// TwinCAT 3 PLC project PLC
// ProgramVersion: 3.1.4024.0
// libraries:
//   EfficientIO ModbusTCP, * (EfficientIO)
//   Lynus Energy Basic, * (Lynus AG)
//   Lynus Persistent Data V1, * (Lynus AG)
//   Lynus Standards, * (Lynus AG)
//   Tc2_IoFunctions, * (Beckhoff Automation GmbH)
//   Tc2_Standard, * (Beckhoff Automation GmbH)
//   Tc2_System, * (Beckhoff Automation GmbH)
//   Tc3_IotBase, * (Beckhoff Automation GmbH)
//   Tc3_IPCDiag, * (Beckhoff Automation GmbH)
//   Tc3_Module, * (Beckhoff Automation GmbH)
// project tree:
//   / FastTask.TcTTO, MiddleTask.TcTTO, SlowTask.TcTTO
//   POUs/ prgComEffIO.TcPOU (excluded from build), prgComEffIO_1.TcPOU (excluded from build), prgEM.TcPOU, prgRWEffIO.TcPOU (not stored) (excluded from build), prgRWEffIO_1.TcPOU (excluded from build), prgTemperature.TcPOU, prgVarEffIO.TcPOU (not stored) (excluded from build), prgVarEffIO_1.TcPOU (excluded from build)
// real-time tasks:
//   TASK PlcTask: cycle T#10ms, priority 20, ADS port 350
//   TASK FastTask: cycle T#5ms, priority 19, ADS port 351
//   TASK MiddleTask: cycle T#10ms, priority 21, ADS port 352
//   TASK SlowTask: cycle T#20ms, priority 23, ADS port 353
// I/O:
//   DEVICE Gerät 2 (CX-BK)
//     Box 1 (CX-BK)
// variable links:
//   PLC/PLC Instance <-> Device 2 (CX-BK)/Box 1 (CX-BK)
//     PlcTask Inputs/prgEM.fbEM1.fbKL3403.byStateCH1 <-> Term 5 (KL3403)/Channel 1/Status
//     PlcTask Inputs/prgEM.fbEM1.fbKL3403.byStateCH2 <-> Term 5 (KL3403)/Channel 2/Status
//     PlcTask Inputs/prgEM.fbEM1.fbKL3403.byStateCH3 <-> Term 5 (KL3403)/Channel 3/Status
//     PlcTask Inputs/prgEM.fbEM1.fbKL3403.iDataInCH1 <-> Term 5 (KL3403)/Channel 1/Daten Ein
//     PlcTask Inputs/prgEM.fbEM1.fbKL3403.iDataInCH2 <-> Term 5 (KL3403)/Channel 2/Daten Ein
//     PlcTask Inputs/prgEM.fbEM1.fbKL3403.iDataInCH3 <-> Term 5 (KL3403)/Channel 3/Daten Ein
//     PlcTask Inputs/prgEM.fbKBusState.uiKBusState_OUT <-> Inputs/State
//     PlcTask Inputs/prgEM.stInData_22/iDataIn <-> Term 4 (KL3204)/Channel 1/Daten Ein
//     PlcTask Inputs/prgEM.stInData_23/iDataIn <-> Term 4 (KL3204)/Channel 2/Daten Ein
//     PlcTask Inputs/prgEM.stInData_22/iState <-> Term 4 (KL3204)/Channel 1/Status
//     PlcTask Inputs/prgEM.stInData_23/iState <-> Term 4 (KL3204)/Channel 2/Status
//     PlcTask Outputs/prgEM.fbEM1.fbKL3403.byCntrCH1 <-> Term 5 (KL3403)/Channel 1/Kontrolle
//     PlcTask Outputs/prgEM.fbEM1.fbKL3403.byCntrCH2 <-> Term 5 (KL3403)/Channel 2/Kontrolle
//     PlcTask Outputs/prgEM.fbEM1.fbKL3403.byCntrCH3 <-> Term 5 (KL3403)/Channel 3/Kontrolle
//     PlcTask Outputs/prgEM.stOutData_22/iCtrl <-> Term 4 (KL3204)/Channel 1/Kontrolle
//     PlcTask Outputs/prgEM.stOutData_23/iCtrl <-> Term 4 (KL3204)/Channel 2/Kontrolle
//     PlcTask Outputs/prgEM.stOutData_22/iDataOut <-> Term 4 (KL3204)/Channel 1/Daten Aus
//     PlcTask Outputs/prgEM.stOutData_23/iDataOut <-> Term 4 (KL3204)/Channel 2/Daten Aus

CONFIGURATION PLC
    RESOURCE PLC ON TwinCAT3
        TASK FastTask(INTERVAL := T#5ms, PRIORITY := 19);
        TASK MiddleTask(INTERVAL := T#10ms, PRIORITY := 21);
        TASK SlowTask(INTERVAL := T#20ms, PRIORITY := 23);
        PROGRAM prgEM WITH MiddleTask : prgEM;
        PROGRAM prgTemperature WITH MiddleTask : prgTemperature;
    END_RESOURCE
END_CONFIGURATION

// ---- POUs/prgEM.TcPOU
PROGRAM prgEM
VAR
	fbKBusState		: FB_K_Bus_State;
	fbEM1			: FB_EM_Beckhoff_KL3403;

END_VAR


fbKBusState(	uiKBusState_OUT=> , 
				b_Kbus_notOk=> , 
				word_ErrorCount=> );
//The mapping OF THIS FUNCTION must be linked with the KL3403 in the E/A Part
// KEBA CS
fbEM1(
	bEnable:= true, 
	bChannel1Invers:= FALSE,				//Invert power data when transformer are mounted upside down
	bChannel2Invers:= FALSE,			
	bChannel3Invers:= FALSE,
	uiCurrentTransformerRatioL1:= 100, //Transformer ratio on the secondary side
	uiCurrentTransformerRatioL2:= 100, 
	uiCurrentTransformerRatioL3:= 100, 
	uiKBusState_IN:= fbKBusState.uiKBusState_OUT, 
	stDataEMPower=> , 
	stDataEMCounter=> , 
	stDataEMPowerRealTime=> , 
	stDataEMCounterRealTime=> , 
	diNrOfEM_OUT=> );

END_PROGRAM

// ---- POUs/prgTemperature.TcPOU
PROGRAM prgTemperature
VAR
// Kanal 1
	fb_Config_1			: FB_KL320xConfig;
	stInData_1   		AT%I*		: ST_KL320xInData;
	stOutData_1		  	AT%Q*		: ST_KL320xOutData;
// Kanal 2
	fb_Config_2			: FB_KL320xConfig;
	stInData_2   		AT%I*		: ST_KL320xInData;
	stOutData_2  		AT%Q*		: ST_KL320xOutData;

END_VAR

	
	
fb_Config_1(
	bConfigurate:= , 
	bReadConfig:= , 
	iSetSensorType:= , 
	tTimeout:= , 
	bBusy=> , 
	bError=> , 
	iErrorId=> , 
	iState=> , 
	iDataIn=> , 
	iTerminalType=> , 
	iSpecialType=> , 
	iFirmwareVersion=> , 
	sDescription=> , 
	sSensorType=> , 
	bTwoWiredConnection=> , 
	stInData:= stInData_1, 
	stOutData:= stOutData_1);
	
fb_Config_2(
	bConfigurate:= , 
	bReadConfig:= , 
	iSetSensorType:= , 
	tTimeout:= , 
	bBusy=> , 
	bError=> , 
	iErrorId=> , 
	iState=> , 
	iDataIn=> , 
	iTerminalType=> , 
	iSpecialType=> , 
	iFirmwareVersion=> , 
	sDescription=> , 
	sSensorType=> , 
	bTwoWiredConnection=> , 
	stInData:= stInData_2, 
	stOutData:= stOutData_2);

END_PROGRAM

// ---- POUs/prgComEffIO.TcPOU
PROGRAM prgComEffIO
VAR
	fbCom		: FB_MqttCommunicator_V2;
	int_PowerLinkNumber: INT;
END_VAR

fbCom(
	bConnect:= TRUE, 
	strAuthkey := 'EIO08031879806',
	sUserName:= '0d7f16f2-b0a8-4684-97E5-cc9fc16b61c5' , 		
	sUserPassword:= '69cd5984-6d64-4e65-aacd-70eb3450ae41',
	eSavePositionCertificate:= eSavePositionOnPLC.ePostionHardDisk, 
	bConnected=> , 
	bError=> , 
	hrErrorCode=> , 
	eConnectionState=> , 
	eErrorMessage_Out=> );

END_PROGRAM

// ---- POUs/prgComEffIO_1.TcPOU
PROGRAM prgComEffIO_1
VAR
	fbCom		: FB_MqttCommunicator_V2;
	int_PowerLinkNumber: INT;
END_VAR

fbCom(
	bConnect:= TRUE, 
	strAuthkey := 'EIO08031879806',
	sUserName:= '0d7f16f2-b0a8-4684-97E5-cc9fc16b61c5' , 		
	sUserPassword:= '69cd5984-6d64-4e65-aacd-70eb3450ae41',
	eSavePositionCertificate:= eSavePositionOnPLC.ePostionHardDisk, 
	bConnected=> , 
	bError=> , 
	hrErrorCode=> , 
	eConnectionState=> , 
	eErrorMessage_Out=> );

END_PROGRAM

// ---- POUs/prgRWEffIO_1.TcPOU
PROGRAM prgRWEffIO_1
VAR
	fbRW1		: FB_ReadWrite_V2;
END_VAR

fbRW1(eUploadType := eSelectDataUploadType.e_Change_Intervall5min, bBusy=> , bError=> , udiErrorCodeOut=> , eErrorReadWrite_Out=> );

END_PROGRAM

// ---- POUs/prgVarEffIO_1.TcPOU
PROGRAM prgVarEffIO_1
VAR
	fbVar		: FB_VarInfo;
END_VAR

fbVar(
	bReadInfo:= , 
	eTMCFile:= eSelectTMCFile.eDontUseTMCFile, 
	eSavePositionTMCFile:= eSavePositionOnPLC.ePostionHardDisk, 
	udiCounterFoundVariables=> , 
	bError=> , 
	bBusy=> , 
	byProgress=> , 
	udiErrorCodeOut=> , 
	eErrorVarInfo_Out=> , 
	sVarWithError=> );

END_PROGRAM
